(* PLC project Unnamed, Unknown Unnamed 1 *)
(* stored: creationDateTime 2026-01-03T09:22:32, modificationDateTime 2026-01-03T09:22:32 *)

PROGRAM main
  VAR
    ButtonON_LED AT %IX100.0 : BOOL;
    ButtonOFF_LED AT %IX100.1 : BOOL;
    ButtonON_LEDBlink AT %IX100.2 : BOOL;
    ButtonOFF_LEDBlink AT %IX100.3 : BOOL;
    LED1 AT %QX100.0 : BOOL;
    LED2 AT %QX100.1 : BOOL;
    LED3 AT %QX100.2 : BOOL;
  END_VAR
  VAR
    Start_Blink : BOOL;
    TON0_Coil : BOOL;
    TON1_Coil : BOOL;
    TON0 : TON;
    TON1 : TON;
  END_VAR

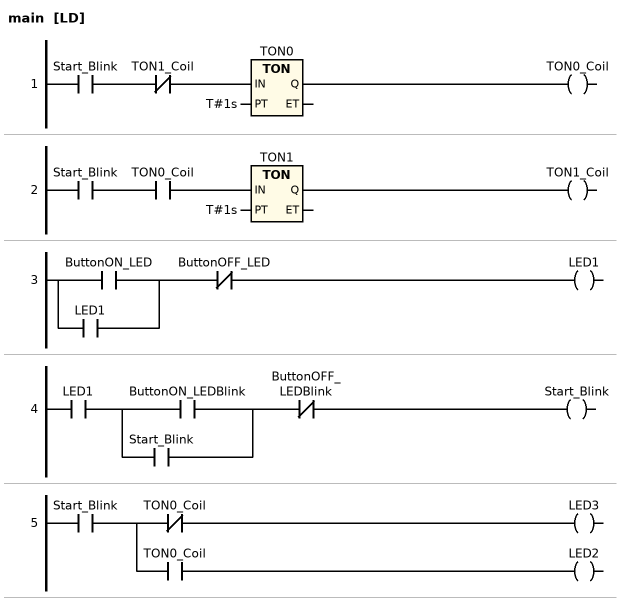
(* LD diagram, written out as Structured Text *)
LED1 := (ButtonON_LED OR LED1) AND NOT ButtonOFF_LED;
Start_Blink := LED1 AND (ButtonON_LEDBlink OR Start_Blink) AND NOT ButtonOFF_LEDBlink;
TON0(IN := Start_Blink AND NOT TON1_Coil, PT := T#1s);
TON0_Coil := TON0.Q;
TON1(IN := Start_Blink AND TON0_Coil, PT := T#1s);
TON1_Coil := TON1.Q;
LED3 := Start_Blink AND NOT TON0_Coil;
LED2 := Start_Blink AND TON0_Coil;
END_PROGRAM

CONFIGURATION Config0
  RESOURCE Res0 ON PLC
    TASK task0(INTERVAL := T#20ms, PRIORITY := 1);
    PROGRAM instance0 WITH task0 : main;
  END_RESOURCE
END_CONFIGURATION
